FUNCTION_BLOCK LED_UBI_MQTT
  {SET_ATTRIBUTE(OpcUa, SERVICE)}
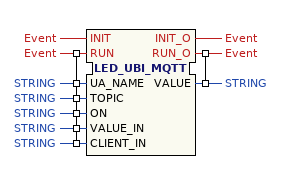
  EVENT_INPUT
    INIT;
    RUN WITH UA_NAME, TOPIC, ON, VALUE_IN, CLIENT_IN;
  END_EVENT
  EVENT_OUTPUT
    INIT_O;
    RUN_O WITH VALUE;
  END_EVENT
  VAR_INPUT
    UA_NAME : STRING; {SET_ATTRIBUTE(OpcUa, Constant)}
    TOPIC : STRING; {SET_ATTRIBUTE(OpcUa, Constant)}
    ON : STRING; {SET_ATTRIBUTE(OpcUa, Constant)}
    VALUE_IN : STRING; {SET_ATTRIBUTE(OpcUa, Variable)}
    CLIENT_IN : STRING; {SET_ATTRIBUTE(OpcUa, Variable)}
  END_VAR
  VAR_OUTPUT
    VALUE : STRING; {SET_ATTRIBUTE(OpcUa, Variable)}
  END_VAR
END_FUNCTION_BLOCK
